// TIA Portal project "Acionamento motor de passo" (V17)
// Testes no desenvolvimento do acionamento motor de passo.

(* hardware
DEVICE "S7-1200 station_1"  S7-1200 Station
   slot 0: "Rack_0"  S7-1200 Rack  Rack  V1.0
   slot 1: "PLC_1"  CPU 1214C DC/DC/DC  6ES7 214-1AG40-0XB0  V4.5
DEVICE "HMI_1"  KTP700 Basic PN
   slot 0: "HMI_1"  KTP700 Basic PN  6AV2 123-2GB03-0AX0  17.0.0.0
   slot 1: "HMI_RT_1"  KTP700 Basic PN  6AV2 123-2GB03-0AX0  17.0.0.0
   slot 5: "HMI_1.IE_CP_1"  PROFINET Interface  17.0.0.0
      slot 1: "PROFINET Interface_1"  PROFINET Interface
         slot 1: "Port_1"  Port
*)

// ===== PLC "PLC_1"  CPU 1214C DC/DC/DC =====

VAR_GLOBAL   // PLC tag table "Default tag table"
   "liga" AT %I0.0 : Bool;
   "liga2" AT %I0.1 : Bool;
   "mliga" AT %M0.0 : Bool;
   "PWM" AT %MB1008 : Byte;
   "PWM(1)" AT %QW1000 : Word;
   "duty_ciclo" AT %MD2 : Real;
   "ciclo(%)" AT %MD6 : Real;
   "Clock_Byte" AT %MB100 : Byte;
   "Clock_10Hz" AT %M100.0 : Bool;
   "Clock_5Hz" AT %M100.1 : Bool;
   "Clock_2.5Hz" AT %M100.2 : Bool;
   "Clock_2Hz" AT %M100.3 : Bool;
   "Clock_1.25Hz" AT %M100.4 : Bool;
   "Clock_1Hz" AT %M100.5 : Bool;
   "Clock_0.625Hz" AT %M100.6 : Bool;
   "Clock_0.5Hz" AT %M100.7 : Bool;
   "reset" AT %M0.1 : Bool;
   "count" AT %MW28 : Int;
   "tempoCount" AT %MW14 : Int;
   "hantiHorario" AT %M0.2 : Bool;
   "direcao" AT %Q0.1 : Bool;
   "habilitaDrive" AT %M0.3 : Bool;
   "driveHabilita" AT %Q0.2 : Bool;
   "habilita_PWM_auto" AT %M0.4 : Bool;
   "habilita_PWM_manu" AT %M0.5 : Bool;
   "habilita_Pulso" AT %M0.6 : Bool;
   "tempoPulso" AT %MD16 : Time;
   "pulsoAlto" AT %M0.7 : Bool;
   "pulsoBaixo" AT %M1.0 : Bool;
   "pulso_drive_motor" AT %Q0.0 : Bool;
   "teste" AT %MD20 : Real;
   "habilitaBloco" AT %M1.1 : Bool;
   "frequencia" AT %MD24 : UDInt;
   "count1" AT %MW10 : Int;
   "sensor" AT %I0.2 : Bool;
END_VAR

DATA_BLOCK "Data_block_1"   // DB4
{ S7_Optimized_Access := 'TRUE' }
VERSION : 0.1
   VAR
      teste_dutyCiclo : Int := 50;
   END_VAR
   VAR RETAIN
      frequencia : UDInt := 100;
   END_VAR
BEGIN
END_DATA_BLOCK

// folder: System blocks/Program resources

DATA_BLOCK "IEC_Counter_0_DB"   // DB1
{ S7_Optimized_Access := 'TRUE' }
AUTHOR : Simatic
FAMILY : IEC
NAME : CNTR
VERSION : 1.0
// stored: InstanceOfName IEC_COUNTER
"IEC_COUNTER"
BEGIN
END_DATA_BLOCK

DATA_BLOCK "timer_01"   // DB3
{ S7_Optimized_Access := 'TRUE' }
AUTHOR : Simatic
FAMILY : IEC
NAME : IEC_TMR
VERSION : 1.0
// stored: InstanceOfName IEC_TIMER
"IEC_TIMER"
BEGIN
END_DATA_BLOCK

// folder: (top level)

FUNCTION "PWM_MANUAL" : Void   // FC1, LAD
{ S7_Optimized_Access := 'TRUE' }
VERSION : 0.1
BEGIN

REGION Network 1
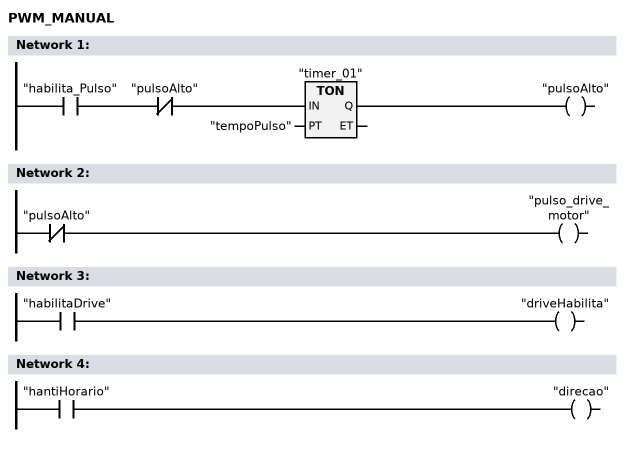
   "timer_01".TON(IN := "habilita_Pulso" AND NOT "pulsoAlto", PT := "tempoPulso");
   "pulsoAlto" := "timer_01".Q;
END_REGION

REGION Network 2
   RUNG wire#powerrail
      I_Contact( "pulsoAlto" )
      Coil( "pulso_drive_motor" )
   END_RUNG
   // the same network as SCL:
   "pulso_drive_motor" := NOT "pulsoAlto";
END_REGION

REGION Network 3
   RUNG wire#powerrail
      Contact( "habilitaDrive" )
      Coil( "driveHabilita" )
   END_RUNG
   // the same network as SCL:
   "driveHabilita" := "habilitaDrive";
END_REGION

REGION Network 4
   RUNG wire#powerrail
      Contact( "hantiHorario" )
      Coil( "direcao" )
   END_RUNG
   // the same network as SCL:
   "direcao" := "hantiHorario";
END_REGION
END_FUNCTION

FUNCTION "PWM_AUTO" : Void   // FC2, LAD
{ S7_Optimized_Access := 'TRUE' }
VERSION : 0.1
BEGIN

REGION Network 1
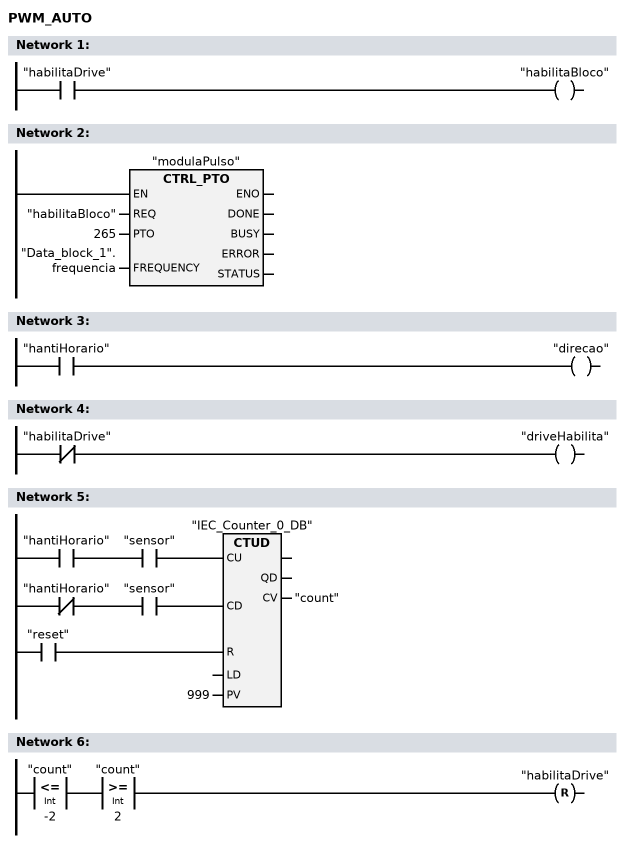
   RUNG wire#powerrail
      Contact( "habilitaDrive" )
      Coil( "habilitaBloco" )
   END_RUNG
   // the same network as SCL:
   "habilitaBloco" := "habilitaDrive";
END_REGION

REGION Network 2
   "modulaPulso"(REQ := "habilitaBloco", PTO := 265, FREQUENCY := "Data_block_1".frequencia);   // CTRL_PTO
END_REGION

REGION Network 3
   RUNG wire#powerrail
      Contact( "hantiHorario" )
      Coil( "direcao" )
   END_RUNG
   // the same network as SCL:
   "direcao" := "hantiHorario";
END_REGION

REGION Network 4
   RUNG wire#powerrail
      I_Contact( "habilitaDrive" )
      Coil( "driveHabilita" )
   END_RUNG
   // the same network as SCL:
   "driveHabilita" := NOT "habilitaDrive";
END_REGION

REGION Network 5
   "IEC_Counter_0_DB".CTUD(CU := "hantiHorario" AND "sensor",
                           CD := NOT "hantiHorario" AND "sensor",
                           R := "reset",
                           PV := 999,
                           CV => "count");
END_REGION

REGION Network 6
   RUNG wire#powerrail
      { S7_Templates := "SrcType := Int" } LE_Contact(in1 := "count", in2 := -2)
      { S7_Templates := "SrcType := Int" } GE_Contact(in1 := "count", in2 := 2)
      R_Coil( "habilitaDrive" )
   END_RUNG
   // the same network as SCL:
   IF ("count" <= (-2)) AND ("count" >= 2) THEN "habilitaDrive" := FALSE; END_IF;
END_REGION
END_FUNCTION

ORGANIZATION_BLOCK "Main"   // OB1, LAD, ProgramCycle
TITLE = "Main Program Sweep (Cycle)"
{ S7_Optimized_Access := 'TRUE' }
VERSION : 0.1
   VAR_INPUT
      Initial_Call : Bool;   // Initial call of this OB
      Remanence : Bool;   // =True, if remanent data are available
   END_VAR
BEGIN

REGION Network 1
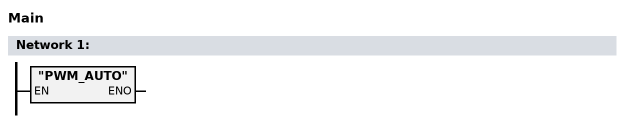
   RUNG wire#powerrail
      "PWM_AUTO"()
   END_RUNG
   // the same network as SCL:
   "PWM_AUTO"();
END_REGION
END_ORGANIZATION_BLOCK

(* ===== HMI "HMI_RT_1" =====
system functions are stored by id; their names below are inferred from use
connection "HMI_Connection_1": ETHERNET, SMART_S7_1200_OMS

HMI tags "Default tag table"
   "teste" : Real = PLC teste AT %MD20, 1 s
   "Data_block_1_frequencia" : UDInt = PLC Data_block_1.frequencia, 1 s
   "habilitaDrive" : Bool = PLC habilitaDrive AT %M0.3, 1 s
   "hantiHorario" : Bool = PLC hantiHorario AT %M0.2, 1 s

screen "Root screen" 800x480, template "Template_1"
   TextField "HmiScreenItemData" at 80,225 size 640x25; Text 'Welcome to HMI_1 (KTP700 Basic+ PN)!'
   IOField "I/O field_1" at 49,60 size 96x32; FormatPattern 9999
      ProcessValue <- "Data_block_1_frequencia"
   Button "Button_1" at 49,117 size 96x32; TextOff 'Liga'
      on Release: SetBit("habilitaDrive")
   Button "Button_2" at 49,167 size 96x32; TextOff 'Desliga'
      on Release: ResetBit("habilitaDrive")
   Button "Button_3" at 49,225 size 96x32; TextOff 'Abre'
      on Release: SetBit("hantiHorario")
   Button "Button_4" at 49,279 size 96x32; TextOff 'Fecha'
      on Release: ResetBit("hantiHorario")
*)